FUNCTION_BLOCK INITswitch
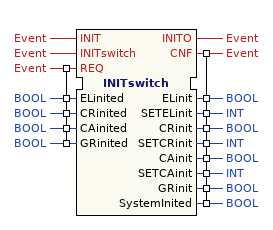
  EVENT_INPUT
    INIT;
    INITswitch;
    REQ WITH ELinited, CRinited, CAinited, GRinited;
  END_EVENT
  EVENT_OUTPUT
    INITO;
    CNF WITH ELinit, SETELinit, CRinit, SETCRinit, CAinit, SETCAinit, GRinit, SystemInited;
  END_EVENT
  VAR_INPUT
    ELinited : BOOL;
    CRinited : BOOL;
    CAinited : BOOL;
    GRinited : BOOL;
  END_VAR
  VAR_OUTPUT
    ELinit : BOOL;
    SETELinit : INT;
    CRinit : BOOL;
    SETCRinit : INT;
    CAinit : BOOL;
    SETCAinit : INT;
    GRinit : BOOL;
    SystemInited : BOOL;
  END_VAR
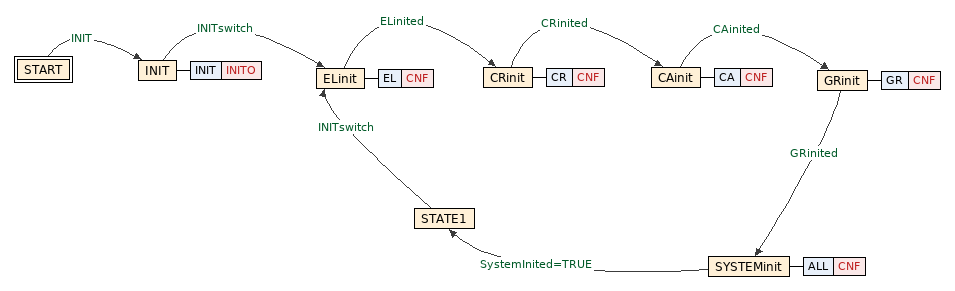
  EC_STATES
    START;
    INIT : INIT -> INITO;
    ELinit : EL -> CNF;
    CRinit : CR -> CNF;
    CAinit : CA -> CNF;
    GRinit : GR -> CNF;
    SYSTEMinit : ALL -> CNF;
    STATE1;
  END_STATES
  EC_TRANSITIONS
    START TO INIT := INIT;
    INIT TO ELinit := INITswitch;
    ELinit TO CRinit := ELinited;
    CRinit TO CAinit := CRinited;
    CAinit TO GRinit := CAinited;
    GRinit TO SYSTEMinit := GRinited;
    SYSTEMinit TO STATE1 := SystemInited=TRUE;
    STATE1 TO ELinit := INITswitch;
  END_TRANSITIONS
  ALGORITHM INIT IN ST:
CAinit := FALSE;
CRinit := FALSE;
ELinit := FALSE;
GRinit := FALSE;
SystemInited := FALSE;
  END_ALGORITHM
  ALGORITHM EL IN ST:
ELinit := TRUE;
SETELinit := 0;
CAinit := FALSE;
CRinit := FALSE;
GRinit := FALSE;
  END_ALGORITHM
  ALGORITHM CR IN ST:
CRinit := TRUE;
SETCRinit := 0;
CAinit := FALSE;
ELinit := FALSE;
GRinit := FALSE;
  END_ALGORITHM
  ALGORITHM CA IN ST:
CAinit := TRUE;
SETCAinit := 1;
CRinit := FALSE;
ELinit := FALSE;
GRinit := FALSE;
  END_ALGORITHM
  ALGORITHM GR IN ST:
GRinit := TRUE;
CAinit := FALSE;
CRinit := FALSE;
ELinit := FALSE;
  END_ALGORITHM
  ALGORITHM ALL IN ST:
SystemInited := TRUE;
CAinit := FALSE;
CRinit := FALSE;
ELinit := FALSE;
GRinit := FALSE;
  END_ALGORITHM
END_FUNCTION_BLOCK
